TYPE GForceMeasurementStatuses :
STRUCT
	///Is the measurement OK?
	healthStatus: HealthStatus;
END_STRUCT
END_TYPE

(* stored: Version 1.1.0.1, ProductVersion 3.1.4019.2
   DUT GForceMeasurementStatuses: Id {2ed5ef7e-41e0-42c7-ac2c-5776c4f0acdb} *)
